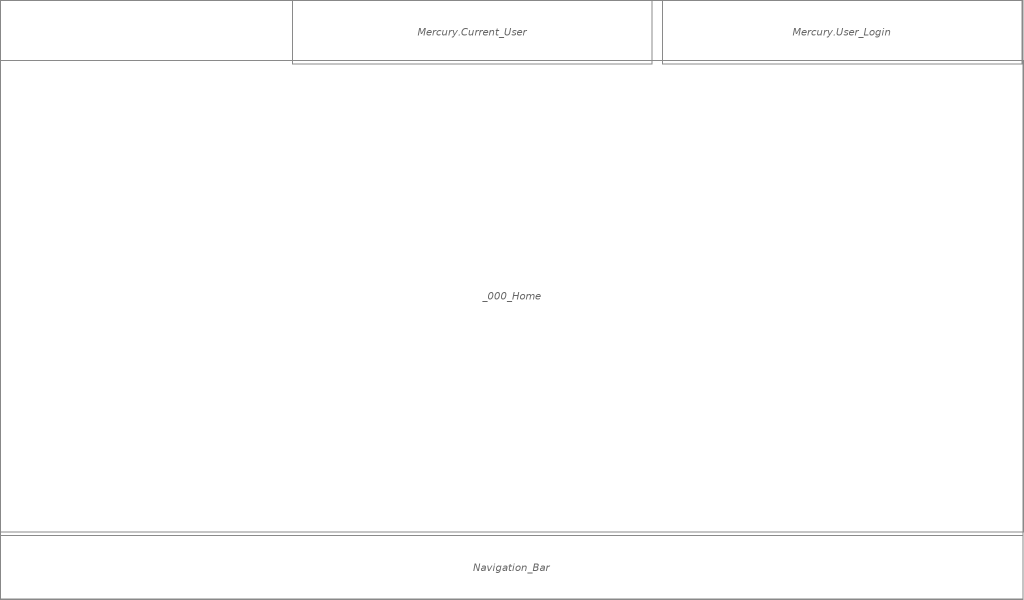
VISUALIZATION FP  // 1024x600, background image JMTC.Swindon_Glovebox_UI_Background
    Frame (0,535 1023x65)
        shows Navigation_Bar()
    Frame (292,0 360x64)
        shows Mercury.Current_User()
    Frame (662,0 360x64), invisible if: HgV_Engine.stNav_Button[3].bInvisible
        shows Mercury.User_Login()
    Frame (0,60 1024x472), frame switch variable: HgV_Engine.propCurrent_Page_
        shows _000_Home()
        shows _001_Blank_1()
        shows _002_Blank_2()
        shows _003_Settings()
END_VISUALIZATION

(* stored: Version 1.1.0.1, ProductVersion 3.1.4022.18
   Visu FP: Id {909a3e92-7cce-4911-952b-c6d88410851f} *)
